// TIA Portal V20 export
DATA_BLOCK "dGlobal"   // DB30150
{ S7_Optimized_Access := 'TRUE' }
// stored: AutoNumber false, MemoryReserve 100
   VAR
      gbo_Axis_Select { S7_SetPoint := 'True'} : Int;
      gbo_Pos_Select : Int;
      gto_Axis_Name : Array[0..9] of DB_ANY;
      gto_Axis_Index : DB_ANY;
      gr64_Pos_Index : LReal;
      Old_Axis_Select : Int;
      Old_Pos_Select : Int;
      gbo_Fault_Reset : Bool;
   END_VAR
   VAR RETAIN
      gi_Axis_AbsNum : Array[0..9] of Int;
   END_VAR
   VAR
      gbo_Axis_ManEnable : Array[0..9] of Bool;
   END_VAR
BEGIN
   gi_Axis_AbsNum[0] := 5;
   gi_Axis_AbsNum[1] := 6;
   gi_Axis_AbsNum[2] := 10;
   gi_Axis_AbsNum[3] := 5;
   gi_Axis_AbsNum[4] := 6;
   gi_Axis_AbsNum[5] := 7;
   gi_Axis_AbsNum[6] := 8;
   gi_Axis_AbsNum[7] := 9;
   gi_Axis_AbsNum[8..9] := 5;
   gbo_Axis_ManEnable[0..9] := 1;
END_DATA_BLOCK
